(* IEC 61131-3 sources: SIGMATEK-Jumag-Utils-Examples/timeConversion/Class/Class0, 1 file *)

(* ---- Class0.st ---- *)
(*!
<Class
	Name               = "Class0"
	Revision           = "0.0"
	RealtimeTask       = "false"
	CyclicTask         = "true"
	DefCyclictime      = "10 ms"
	BackgroundTask     = "false"
	Sigmatek           = "false"
	OSInterface        = "false"
	HighPriority       = "false"
	Automatic          = "false"
	UpdateMode         = "Prescan"
	SharedCommandTable = "true"
	Objectsize         = "(284,120)">
	<Channels>
		<Server Name="ClassSvr" Visualized="false" Initialize="false" WriteProtected="true" Retentive="false"/>
		<Server Name="convertedToMinutes" Visualized="false" Initialize="false" WriteProtected="true" Retentive="false"/>
		<Server Name="convertedToSeconds" Visualized="false" Initialize="false" WriteProtected="true" Retentive="false"/>
		<Server Name="unconvertedMillis" Visualized="false" Initialize="false" WriteProtected="false" Retentive="false"/>
	</Channels>
	<Dependencies>
		<Files>
			<File Path=".\Source\timeConversion.c"/>
		</Files>
	</Dependencies>
</Class>
*)
Class0 : CLASS
  //Servers:
	ClassSvr 	: SvrChCmd_DINT;
	unconvertedMillis 	: SvrCh_UDINT;
	convertedToSeconds 	: SvrCh_UDINT;
	convertedToMinutes 	: SvrCh_UDINT;
  //Clients:
  //Variables:
  //Functions:

	FUNCTION VIRTUAL GLOBAL CyWork
		VAR_INPUT
			EAX 	: UDINT;
		END_VAR
		VAR_OUTPUT
			state (EAX) 	: UDINT;
		END_VAR;
  //Tables:
	FUNCTION @STD
		VAR_OUTPUT
			ret_code	: CONFSTATES;
		END_VAR;
	FUNCTION GLOBAL TAB @CT_;
END_CLASS;

Function Global __cdecl ms_to_s
VAR_INPUT
  millis : UDINT;
END_VAR
VAR_OUTPUT
  seconds : UDINT;
END_VAR;

Function Global __cdecl ms_to_min
VAR_INPUT
  millis : UDINT;
END_VAR
VAR_OUTPUT
  minutes : UDINT;
END_VAR;

FUNCTION VIRTUAL GLOBAL Class0::CyWork
	VAR_INPUT
		EAX 	: UDINT;
	END_VAR
	VAR_OUTPUT
		state (EAX) 	: UDINT;
	END_VAR

	state := READY;
  unconvertedMillis := ops.tAbsolute;

  convertedToSeconds := ms_to_s(millis:=unconvertedMillis);
  convertedToMinutes := ms_to_min(millis:=unconvertedMillis);

END_FUNCTION
